Staubli VAL3: midPos.pgx

public program midPos(string x_sItem, num x_nLenght, num x_nPos, string& x_sResult[])
  local string l_sLeft
begin
  // LEFT SIDE
  call leftPos(x_sItem,x_nLenght+x_nPos,l_sLeft)
  // update
  x_sResult=l_sLeft
  // RIGHT SIDE
  call rightPos(l_sLeft,x_nLenght,x_sResult)
  // OK ....
end
